FUNCTION_BLOCK FB_StateMachinePro
VAR_INPUT	
	bEnable : BOOL;
	bStart : BOOL;
	bStop : BOOL;
	
	bBottle : BOOL;				// fotocellula FC1
END_VAR

VAR_OUTPUT
	eStep :  E_Step;
	tStepTime : TIME;
	eErrStep : E_Step;
	nErrId : DINT;
	
	bConveyor : BOOL;			// nastro trasportatore
	bWater : BOOL;				// riempimento acqua
	bMint : BOOL;				// riempimento menta	
	bCorking : BOOL;			// inserimento del tappo	
END_VAR

VAR_IN_OUT
	
END_VAR

VAR
	bInitialized :  BOOL;
	eNewstep :  E_Step;
	bEntryact :  BOOL;
	fbTonStep :  TON;	
	
	fbTonBottle : TON;
	fbRtBottle : R_TRIG;
	
	fbRtStop : R_TRIG;
	bStopRequest : BOOL;
	
	nFillingCycles : USINT;
END_VAR

IF NOT bInitialized THEN
	eNewstep := E_Step.NoStep;
	eStep := E_Step.Stop;
	bEntryact := FALSE;
	bInitialized := TRUE;		
ELSE	
	(* disabilitata o avaria *)
	IF NOT bEnable THEN
		eNewstep := E_Step.NeOrError;
	END_IF;
	
	IF eNewstep <> E_Step.NoStep THEN
		eStep := eNewstep;
		eNewstep := E_Step.NoStep;
		bEntryact := FALSE;
	END_IF;

	(* filtri *)
	fbTonBottle(IN:= bBottle, PT:= T#500MS);		// filtro sensore presenza bottiglia
	
	(* fronti *)
	fbRtBottle(CLK:= fbTonBottle.Q);
	fbRtStop(CLK:= bStop);
	
	(* richieste *)
	IF fbRtStop.Q THEN
		bStopRequest := TRUE;
	END_IF; 
	
	CASE eStep OF
		
		(* not Enabled or Error *)
		E_Step.NeOrError :
			(* entry action *)
			IF NOT bEntryact THEN
				bEntryact := TRUE;
			END_IF;

			(* body *)
			bConveyor := FALSE;
			bWater := FALSE;
			bMint := FALSE;
			bCorking := FALSE;
			
			nFillingCycles := 0;
					
			(* transition *)
			IF bEnable THEN				
				eNewstep := E_Step.Stop;				
			END_IF;

			(* exitact *)
			IF eNewstep <> E_Step.NoStep THEN
				;
			END_IF;		
			
		(* Stop *)
		E_Step.Stop:
			(* entry action *)
			IF NOT bEntryact THEN
				bStopRequest := FALSE;
				bEntryact := TRUE;
			END_IF;

			(* body *)
			bConveyor := FALSE;
			bWater := FALSE;
			bMint := FALSE;
			bCorking := FALSE;
			
			nFillingCycles := 0;
				
			(* transition *)
			IF bStart THEN
				eNewstep := E_Step.Feeding;
			END_IF
			
			(* exitact *)
			IF eNewstep <> E_Step.NoStep THEN
				;
			END_IF;
			
		(* Feeding *)
		E_Step.Feeding:
			(* entry action *)
			IF NOT bEntryact THEN
				bEntryact := TRUE;
			END_IF;

			(* body *)
			bConveyor := TRUE;
			bWater := FALSE;
			bMint := FALSE;
			bCorking := FALSE;
		
			(* transition *)
			IF bStopRequest AND NOT bBottle THEN
				eNewstep := E_Step.Stopping;
			ELSE
				IF fbRtBottle.Q THEN
					eNewstep := E_Step.WaterFilling;
				END_IF
			END_IF
			
			(* exitact *)
			IF eNewstep <> E_Step.NoStep THEN
				;
			END_IF;
			
		(* Water Filling *)
		E_Step.WaterFilling:
			(* entry action *)
			IF NOT bEntryact THEN
				nFillingCycles := nFillingCycles + 1;
				bEntryact := TRUE;
			END_IF;

			(* body *)
			bConveyor := FALSE;
			bWater := TRUE;
			bMint := FALSE;
			bCorking := FALSE;
		
			(* transition *)
			IF tStepTime >= T#1S500MS THEN
				eNewstep := E_Step.MintFilling;
			END_IF
			
			(* exitact *)
			IF eNewstep <> E_Step.NoStep THEN
				;
			END_IF;
			
		(* Mint Filling *)
		E_Step.MintFilling:
			(* entry action *)
			IF NOT bEntryact THEN
				bEntryact := TRUE;
			END_IF;

			(* body *)
			bConveyor := FALSE;
			bWater := FALSE;
			bMint := TRUE;
			bCorking := FALSE;
		
			(* transition *)
			IF tStepTime >= T#500MS THEN
				IF nFillingCycles >= 3 THEN
					eNewstep := E_Step.Waiting1;
				ELSE 
					eNewstep := E_Step.WaterFilling;
				END_IF
					
			END_IF
			
			(* exitact *)
			IF eNewstep <> E_Step.NoStep THEN
				IF eNewstep = E_Step.Waiting1 THEN
					nFillingCycles := 0;
				END_IF
			END_IF;	

		(* Waiting 1 *)
		E_Step.Waiting1:
			(* entry action *)
			IF NOT bEntryact THEN
				bEntryact := TRUE;
			END_IF;

			(* body *)
			bConveyor := FALSE;
			bWater := FALSE;
			bMint := FALSE;
			bCorking := FALSE;
		
			(* transition *)
			IF tStepTime >= T#1S THEN
				eNewstep := E_Step.Corking;
			END_IF
			
			(* exitact *)
			IF eNewstep <> E_Step.NoStep THEN
				;
			END_IF;	

		(* Corking *)
		E_Step.Corking:
			(* entry action *)
			IF NOT bEntryact THEN
				bEntryact := TRUE;
			END_IF;

			(* body *)
			bConveyor := FALSE;
			bWater := FALSE;
			bMint := FALSE;
			bCorking := TRUE;
		
			(* transition *)
			IF tStepTime >= T#3S THEN
				eNewstep := E_Step.Waiting2;
			END_IF
			
			(* exitact *)
			IF eNewstep <> E_Step.NoStep THEN
				;
			END_IF;

		(* Waiting 2 *)
		E_Step.Waiting2:
			(* entry action *)
			IF NOT bEntryact THEN
				bEntryact := TRUE;
			END_IF;

			(* body *)
			bConveyor := FALSE;
			bWater := FALSE;
			bMint := FALSE;
			bCorking := FALSE;
		
			(* transition *)
			IF tStepTime >= T#1S THEN
				eNewstep := E_Step.Feeding;
			END_IF
			
			(* exitact *)
			IF eNewstep <> E_Step.NoStep THEN
				;
			END_IF;

		(* Stopping *)
		E_Step.Stopping:
			(* entry action *)
			IF NOT bEntryact THEN
				bEntryact := TRUE;
			END_IF;

			(* body *)
			bConveyor := FALSE;
			bWater := tStepTime >= T#200MS AND tStepTime <= T#400MS;
			bMint := tStepTime >= T#200MS AND tStepTime <= T#400MS;
			bCorking := FALSE;
		
			(* transition *)
			IF tStepTime >= T#2S THEN
				eNewstep := E_Step.Stop;
			END_IF; 
			
			(* exitact *)
			IF eNewstep <> E_Step.NoStep THEN
				;
			END_IF;		
		ELSE
			eNewstep := E_Step.NeOrError;
			eErrStep := E_Step.Unknown;
			nErrId := -9;			
	END_CASE;
	
	(* tempo di permanenza nello step *)
	fbTonStep(IN := (eNewstep = E_Step.NoStep), PT := T#500H);
	tStepTime := fbTonStep.ET;
	
END_IF;

END_FUNCTION_BLOCK

(* stored: Version 1.1.0.1, ProductVersion 3.1.4024.12
   POU FB_StateMachinePro: Id {628eea9b-d3a1-4a41-bcf1-9872281aa285}, SpecialFunc None *)
